// LS Electric XG5000 project: timeroff
// PLC LSPLC
// module base 0 slot 0: 입출력 모듈:XBC-DR30S (DC 24V 입력 18점, 릴레이 출력 12점)

PROGRAM timeroff (task: 스캔 프로그램)

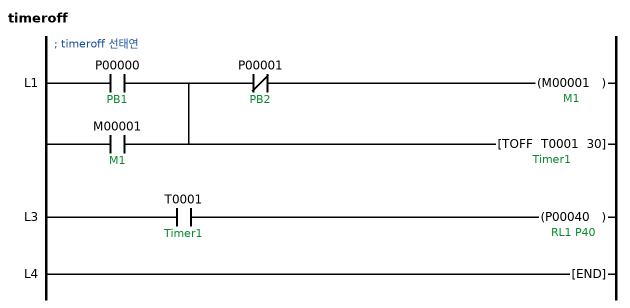
// timeroff 선태연
; L1
LOAD      P00000	// PB1
OR        M00001	// M1
MPUSH
AND NOT   P00001	// PB2
OUT       M00001	// M1
MPOP
TOFF      T0001 30	// Timer1
; L3
LOAD      T0001	// Timer1
OUT       P00040	// RL1 P40
; L4
END